ABB RobotStudio station: Bandeira_20220321-210126.rsstn

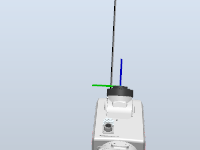
Station Bandeira (saved by RobotStudio 21.4.9700.0)
Controller IRB120_3_58
  mechanical unit ROB_1: IRB120_3_58__01, 6 joints, base frame (0, 0, 0) mm
Layout (positions relative to the parent item):
  - IRB120_3_58__01 [mechanism, from Robots\IRB120_3_58_G_01.rslib] at (0, 0, 0) mm; joint values [-0.0391, 1.3296, -0.4683, -0.0515, -0.8619, 0.0335] (rad or m)
